FUNCTION_BLOCK FB_SubSystem_PMPS_IO
VAR_INPUT
	RequestingSystemID	:	DWORD := PMPS_GVL.EXCLUDED_ASSERTION_ID; // System ID for making requests to the supreme arbiter
    Reset : BOOL;
END_VAR
VAR_OUTPUT
END_VAR
VAR_IN_OUT
	Arbiter	: FB_Arbiter;
    fbFFHWO : FB_HardwareFFOutput;
END_VAR
VAR
	i_RequestedBP AT %I*	:	ST_BeamParams;
	o_CurrentBP AT %Q* : ST_BeamParams;
    
    // EL6692 Diagnostics
    i_Connected AT %I* : BOOL; // SYNC Inputs^External device not connected !!! Doesn't really work.
    i_WcState AT %I* : BOOL; // WcState^WcState
    i_TxPDOState AT %I* : BOOL; // SYNC Inputs^TxPDO state
    
    // Fast faults
    ffPMPSIO_Disconnect : FB_FastFault := (i_Desc:='Fast fault on arbiter disconnection');
END_VAR

// Update arbiter with our request
Arbiter.RemoveRequest(RequestingSystemID);
Arbiter.AddRequest(RequestingSystemID, i_RequestedBP);

// Current beam params fanout
o_CurrentBP := PMPS_GVL.stCurrentBeamParameters;

// Both of these values should be 0 for a fully valid exchange
ffPMPSIO_Disconnect.i_xOK := NOT i_WcState AND NOT i_TxPDOState;

ffPMPSIO_Disconnect(
    io_fbFFHWO := fbFFHWO,
    i_xReset := Reset);

END_FUNCTION_BLOCK

(* stored: Version 1.1.0.1, ProductVersion 3.1.4022.18
   POU FB_SubSystem_PMPS_IO: Id {1a7d9761-dced-4384-823d-a5e0b037bf80}, SpecialFunc None *)
